FUNCTION_BLOCK "G302M_Code"
TITLE =G302M HEATING KILN 2
//COPYRIGHT:    (C) 2009  BUHLER AG, CH-9240 UZWIL, SWITZERLAND
//
//PRODUCT:      WinCoS_BIW01_09
//
//TITLE:        HEATING KILN 2
//                Machine group control
//                Maschinengruppensteuerung
//
//--------------------------------------------------------------------------------
//
//IDENT:        AUTHOR:             DEPT:                              DATE:
//
//P01_FB402.2.0 M.Wedler            AEB41                              27.Apr.2010
//             2nd Release
//P01_FB402.1.0 K.Renz              CSB41                              08.Okt.2009
//             1st Release
//
//--------------------------------------------------------------------------------
//
//PURPOSE:
//
//MANUAL :
//
//RESTRICTIONS:
//
//--------------------------------------------------------------------------------
AUTHOR : KR
FAMILY : USW
VERSION : 9.9


VAR
  Gr : "GCS7_GrpCtrlSub";	//Standard interface to group
  InOutValue1 : DINT ;	//Data for user
  InOutValue2 : DINT ;	//Data for user
  OutWayConflict : BOOL ;	//Data for user
  OutSelectionOk : BOOL ;	//Data for user
  CmdNewValue : BOOL ;	//Data for user
  CmdNewJob : BOOL ;	//Data for user
  OutCodeOK : BOOL ;	//Data for user
  InEndOfJob : BOOL ;	//Data for user
  staWayOk : BOOL ;	//Data for user
  EdgeStartRelease : BOOL ;	//Data for user
  USW8 : BOOL ;	//Data for user
  USW9 : BOOL ;	//Data for user
  USW10 : BOOL ;	//Data for user
  USW11 : BOOL ;	//Data for user
  USW12 : BOOL ;	//Data for user
  USW13 : BOOL ;	//Data for user
  USW14 : BOOL ;	//Data for user
  USW15 : BOOL ;	//Data for user
  A_3291_BPS21 : "GCS7_E_DigInput";	// DigInpCont
  A_3261_KCL11 : "GCS7_E_DigInput";	// DigInpCont
  A_3261_KCL11_AI : "GCS7_E_AnalogInput";	// AnaInp
  A_3261_KCL11_AO : "GCS7_E_AnalogOutput";	// AnaOutp
  A_3261_KCL11_EXT_ON : "GCS7_E_DigOutput";	// DigOut
  A_3261_KCL11_ON : "GCS7_E_DigInput";	// DigInpCont
  A_3261_KCL11_RUN : "GCS7_E_DigOutput";	// DigOut
  A_3261_KCL11_REG_ON : "GCS7_E_DigInput";	// DigInpCont
  A_3261_KCL11_REM_OP : "GCS7_E_DigInput";	// DigInpCont
END_VAR
VAR_TEMP
  tmpEnable : BOOL ;
  tmpFlag : BOOL ;
  tmpCmdNext : BOOL ;
  tmpLocal : BOOL ;
  tmpAspOk : BOOL ;
  tmpHWStop : BOOL ;
  tmpInstanzDBNo : INT ;
END_VAR
BEGIN
NETWORK
TITLE =



NETWORK
TITLE =Read command from group control
//Parameter
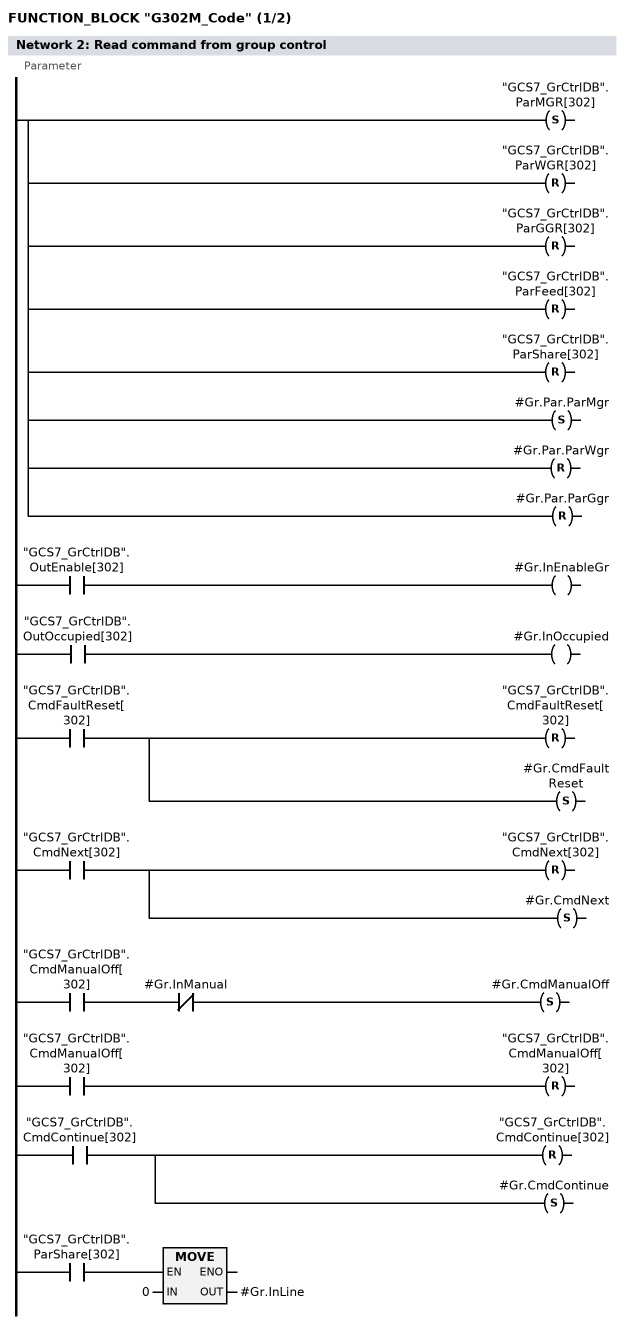
      SET   ;
      S     "GCS7_GrCtrlDB".ParMGR[302];
      R     "GCS7_GrCtrlDB".ParWGR[302];
      R     "GCS7_GrCtrlDB".ParGGR[302];
      R     "GCS7_GrCtrlDB".ParFeed[302];
      R     "GCS7_GrCtrlDB".ParShare[302];
      S     #Gr.Par.ParMgr;
      R     #Gr.Par.ParWgr;
      R     #Gr.Par.ParGgr;
//Command
      U     "GCS7_GrCtrlDB".OutEnable[302];
      =     #Gr.InEnableGr;
      U     "GCS7_GrCtrlDB".OutOccupied[302];
      =     #Gr.InOccupied;
      U     "GCS7_GrCtrlDB".CmdFaultReset[302];
      R     "GCS7_GrCtrlDB".CmdFaultReset[302];
      S     #Gr.CmdFaultReset;
      U     "GCS7_GrCtrlDB".CmdNext[302];
      R     "GCS7_GrCtrlDB".CmdNext[302];
      S     #Gr.CmdNext;

      U     "GCS7_GrCtrlDB".CmdManualOff[302];
      UN    #Gr.InManual;
      S     #Gr.CmdManualOff;
      U     "GCS7_GrCtrlDB".CmdManualOff[302];
      R     "GCS7_GrCtrlDB".CmdManualOff[302];

//      U     "GCS7_GrCtrlDB".CmdManualOff[302]
//      O     "GCS7_GrCtrlDB".OutOccupied[302]
//      R     "GCS7_GrCtrlDB".CmdManualOff[302]
//      S     #Gr.CmdManualOff

      U     "GCS7_GrCtrlDB".CmdContinue[302];
      R     "GCS7_GrCtrlDB".CmdContinue[302];
      S     #Gr.CmdContinue;
//Init Line Number
      U     "GCS7_GrCtrlDB".ParShare[302];
      SPBN  WE00;
      L     0;
      T     #Gr.InLine;
WE00: NOP   0;
NETWORK
TITLE =Call Methode Control
// 1. Handle Interface PCControl
// 2. Prepare mode --> ModePassive,ModeActive,ModeIdling
// 3. Reset global flags of the group
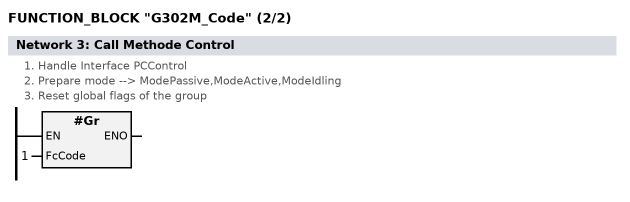
      CALL #Gr (
           FcCode                   := 1);
NETWORK
TITLE =Restart Idling Time

      L     #Gr.Par.ParIdling;
      L     2;
      >=I   ;
      SPB   IdTm;
      T     #Gr.Par.ParIdling;
IdTm: NOP   0;
      CLR   ;
      S     #Gr.CmdRestartIdling;
NETWORK
TITLE =Prepare global flags



NETWORK
TITLE =Set Pattern (Target position)

      U     #Gr.InManual;
      SPB   ILO6;
      L     "MAL1S033Par".StepAct.TemperaturBelowFloor;
      L     L#10;
      /D    ;
      DTR   ;
      U     "MAL1S033Par".Par.FlagProcess.Inf08; // Schritt halten
      SPBN  En06;
      L     "MAL1S033Par".RecipeHeader.SPARE_INT001; // Temp aus General Rezept
      DTR   ;
      SPA   En06;
ILO6: NOP   0;
      L     "MAL1S033Par".Par.ParIntProcess.TargetTemperature_ILO;
      ITD   ;
      DTR   ;
En06: T     "Regler Brenner 3".SP_INT; // setpoint temperature


NETWORK
TITLE =Interlocking WayOk

//BRT20100830 ====> Schritt abhängig den Abschaltpunkt für Brenner verändern
      U     "MAL1S033Par".Par.FlagProcess.ProcessActive;
      U(    ;
      L     "MAL1S033Par".Par.ParIntMachine.ActualStep;
      L     3;
      <I    ;
      )     ;
      U     "MAL1S032Par".Par.FlagProcess.Abdarr_Betrieb_Aktiv;
      L     "MAL1S033Par".StepAct.TemperaturBelowFloor;
      L     30;
      +I    ;
      L     10;
      *I    ;
      SPB   dif1;
      L     "MAL1S033Par".StepAct.TemperaturBelowFloor;
      L     100; // 10,0°C mehr als Sollwert
      +I    ;
      L     10;
      *I    ;
dif1: T     #InOutValue1; // Schaltpunkt für Brenner OFF

      U     "MAL1S033Par".Par.FlagProcess.ProcessActive;
      U(    ;
      L     "MAL1S033Par".Par.ParIntMachine.ActualStep;
      L     3;
      <I    ;
      )     ;
      U     "MAL1S032Par".Par.FlagProcess.Abdarr_Betrieb_Aktiv;
      L     "MAL1S033Par".StepAct.TemperaturBelowFloor;
      L     20;
      -I    ;
      L     10;
      *I    ;
      SPB   dif2;
      L     "MAL1S033Par".StepAct.TemperaturBelowFloor;
      L     10;
      *I    ;
dif2: T     #InOutValue2; // Schaltpunkt für Brenner ON


// Switch "OFF" Burner by Over Temperature
      U     "MAL1S033Par".Par.FlagProcess.ProcessActive;
      U(    ;
//      L     "MAL1S033Par".StepAct.TemperaturBelowFloor
//      L     100                         // 5,0°C mehr als Sollwert
//      +I
//      L     10
//      *I
      L     #InOutValue1; // Schaltpunkt für Brenner OFF
      L     "G295M".A_3291_BTE01.OutValuePc; //  Temperature Below Kiln Floor
      <=I   ;
      )     ;
      S     "G302M".USW8; //Over Temperature

      U(    ;
//      L     "MAL1S033Par".StepAct.TemperaturBelowFloor
//      L     10
//      *I
      L     #InOutValue2; // Schaltpunkt für Brenner ON
      L     "G295M".A_3291_BTE01.OutValuePc; //  Temperature Below Kiln Floor
      >=I   ;
      )     ;
      ON    "MAL1S033Par".Par.FlagProcess.ProcessActive;
      R     "G302M".USW8; //Over Temperature

//BRT20100830 <====
NETWORK
TITLE =Interlocking Autostart

      CLR   ;
      R     #Gr.OutAutostart;
NETWORK
TITLE =Interlocking Enable
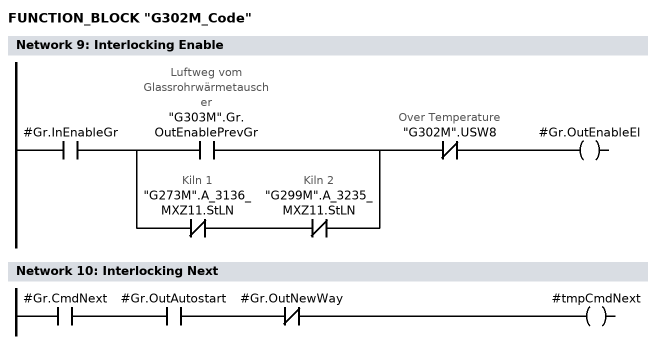

      U     #Gr.InEnableGr;
      U(    ;
      U     "G303M".Gr.OutEnablePrevGr; // Luftweg vom Glassrohrwärmetauscher
      O     ; // Umluftkanal
      UN    "G273M".A_3136_MXZ11.StLN; // Kiln 1
      UN    "G299M".A_3235_MXZ11.StLN; // Kiln 2
      )     ;
      UN    "G302M".USW8; //Over Temperature
      =     #Gr.OutEnableEl;

NETWORK
TITLE =Interlocking Next

      U     #Gr.CmdNext;
      U     #Gr.OutAutostart;
      UN    #Gr.OutNewWay;
      =     #tmpCmdNext;

NETWORK
TITLE =Interlocking Local / HWStop

      U     "PLC_SystemDB".GlobalFlags.Kilning_2;
      CLR   ;
      =     #tmpHWStop;

      U     #Gr.ModePassive;
      O     #tmpHWStop;
      =     #tmpLocal;

NETWORK
TITLE ==A-3291-BPS21 : HEAT EXCHANGE PRESSURE < 15mbar (Reserve)

      NOP   0;
//-InLocal---
      U     #tmpLocal;
      SET   ; // Nur einmal in Darre 1
      =     #A_3291_BPS21.InLocal;
//
//-Monitoring---
      CLR   ;
      =     #A_3291_BPS21.InMonTrue;
      CLR   ;
      =     #A_3291_BPS21.InMonFalse;
//
//-PreAlarm---
      CLR   ;
      =     #A_3291_BPS21.InPreAlarmTrue;
      CLR   ;
      =     #A_3291_BPS21.InPreAlarmFalse;
//
//-Additional commands---
//      CLR
//      S     #A_3291_BPS21.CmdRunTimeOutTime
//
//-Read inputs---
//      U     "A_3291_BPS21_I1"
      CLR   ;
      =     #A_3291_BPS21.InpTrue;
      U     "PLC_SystemDB".GlobalFlags.Kilning_2;
      =     #A_3291_BPS21.InHWStop;
      U     "PLC_DPInfo".Master[1].SlavesError[102];
      =     #A_3291_BPS21.InDPFault;
//
//-Set Parameters---
//
//-Call object control---
      CALL #A_3291_BPS21 ;
//
//-Write outputs---
NETWORK
TITLE ==A-3261-KCL11 : BURNER 3 ALARM SUMMARY

      NOP   0;
//-InLocal---
      U     #tmpLocal;
      =     #A_3261_KCL11.InLocal;
//
//-Monitoring---
      SET   ;
      =     #A_3261_KCL11.InMonTrue;
      CLR   ;
      =     #A_3261_KCL11.InMonFalse;
//
//-PreAlarm---
      CLR   ;
      =     #A_3261_KCL11.InPreAlarmTrue;
      CLR   ;
      =     #A_3261_KCL11.InPreAlarmFalse;
//
//-Additional commands---
//      CLR
//      S     #A_3261_KCL11.CmdRunTimeOutTime
//
//-Read inputs---
      UN    "A_3261_KCL11_I3";
      =     #A_3261_KCL11.InpTrue;
      U     "PLC_SystemDB".GlobalFlags.Kilning_2;
      =     #A_3261_KCL11.InHWStop;
      U     "PLC_DPInfo".Master[1].SlavesError[102];
      =     #A_3261_KCL11.InDPFault;
//
//-Set Parameters---
//
//-Call object control---
      CALL #A_3261_KCL11 ;
//
//-Write outputs---
NETWORK
TITLE ==A-3261-KCL11_EXT_ON : BURNER 3 EXTERAL ON
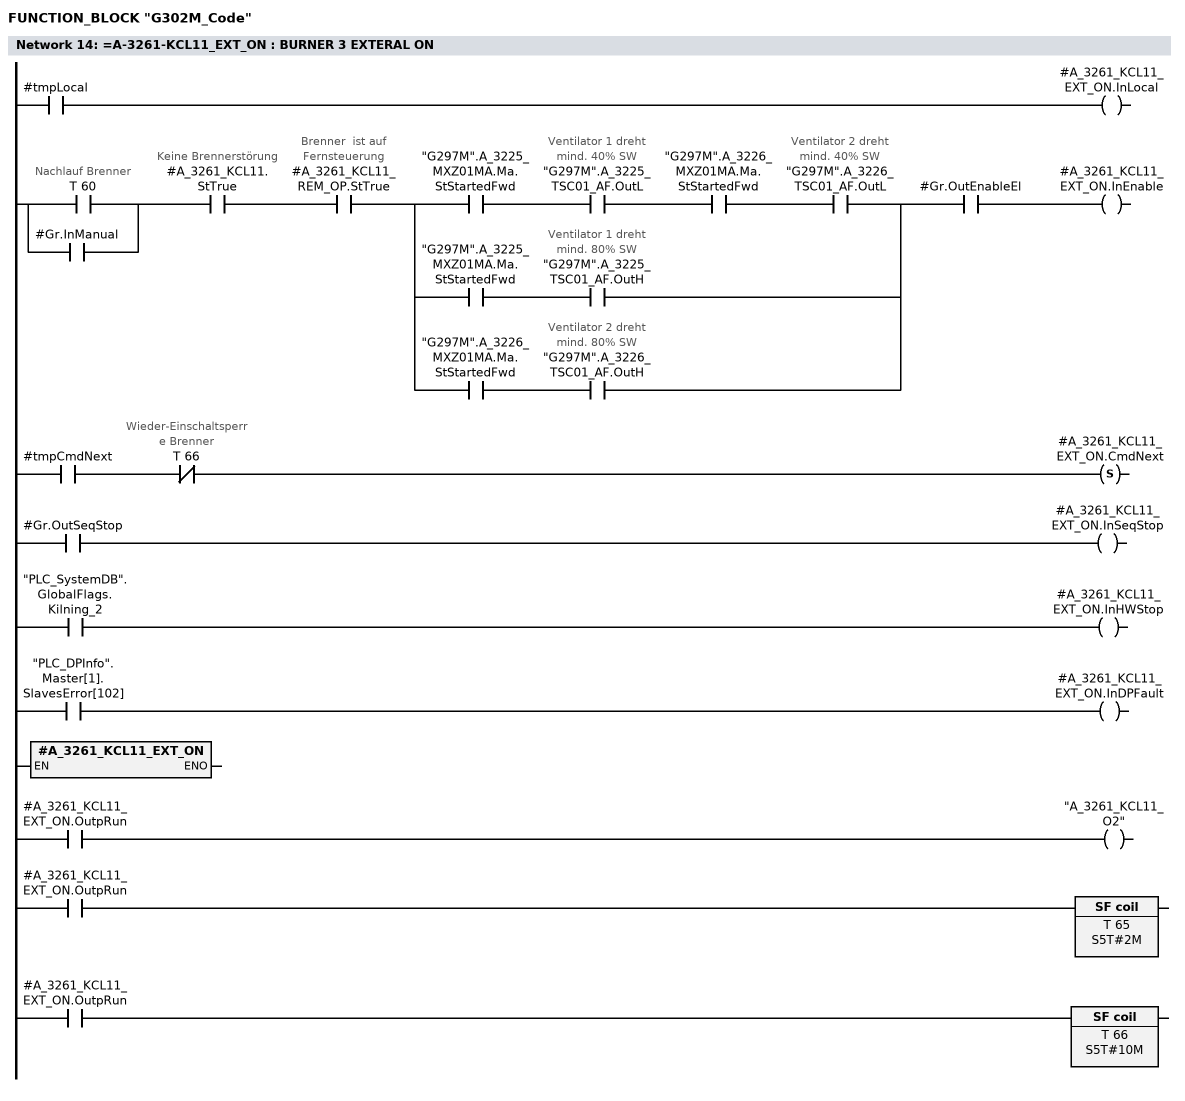

      NOP   0;
//-InLocal---
      U     #tmpLocal;
      =     #A_3261_KCL11_EXT_ON.InLocal;
//
//-Interlocking---
// Signal an Brenner 3: Start
      U     T     60; // Nachlauf Brenner
      O     #Gr.InManual;
      U     #A_3261_KCL11.StTrue; // Keine Brennerstörung
      U     #A_3261_KCL11_REM_OP.StTrue; // Brenner  ist auf Fernsteuerung
      U(    ;
      U     "G297M".A_3225_MXZ01MA.Ma.StStartedFwd;
      U     "G297M".A_3225_TSC01_AF.OutL; // Ventilator 1 dreht mind. 40% SW
      U     "G297M".A_3226_MXZ01MA.Ma.StStartedFwd;
      U     "G297M".A_3226_TSC01_AF.OutL; // Ventilator 2 dreht mind. 40% SW
      O     ;
      U(    ;
      U     "G297M".A_3225_MXZ01MA.Ma.StStartedFwd;
      U     "G297M".A_3225_TSC01_AF.OutH; // Ventilator 1 dreht mind. 80% SW
      O     ;
      U     "G297M".A_3226_MXZ01MA.Ma.StStartedFwd;
      U     "G297M".A_3226_TSC01_AF.OutH; // Ventilator 2 dreht mind. 80% SW
      )     ;
      )     ;
      U     #Gr.OutEnableEl;
      =     #A_3261_KCL11_EXT_ON.InEnable;
//
      U     #tmpCmdNext;
      UN    T     66; // Wieder-Einschaltsperre Brenner
      S     #A_3261_KCL11_EXT_ON.CmdNext;
//
      U     #Gr.OutSeqStop;
      =     #A_3261_KCL11_EXT_ON.InSeqStop;
//
//-Read inputs---
      U     "PLC_SystemDB".GlobalFlags.Kilning_2;
      =     #A_3261_KCL11_EXT_ON.InHWStop;
      U     "PLC_DPInfo".Master[1].SlavesError[102];
      =     #A_3261_KCL11_EXT_ON.InDPFault;
//
//-Set Parameters---
//
//-Call object control---
      CALL #A_3261_KCL11_EXT_ON ;
//
//-Write outputs---
      U     #A_3261_KCL11_EXT_ON.OutpRun;
      =     "A_3261_KCL11_O2";

      U     #A_3261_KCL11_EXT_ON.OutpRun;
      L     S5T#2M;
      SA    T     65; // Nachlauf Ventilator

// Um Stoerungen zu vermeiden
      U     #A_3261_KCL11_EXT_ON.OutpRun;
      L     S5T#10M;
      SA    T     66;

NETWORK
TITLE ==A-3261-KCL11_ON : BURNER 3 ON

      NOP   0;
//-InLocal---
      U     #tmpLocal;
      =     #A_3261_KCL11_ON.InLocal;
//
//-Monitoring---
      CLR   ;
      =     #A_3261_KCL11_ON.InMonTrue;
      CLR   ;
      =     #A_3261_KCL11_ON.InMonFalse;
//
//-PreAlarm---
      CLR   ;
      =     #A_3261_KCL11_ON.InPreAlarmTrue;
      CLR   ;
      =     #A_3261_KCL11_ON.InPreAlarmFalse;
//
//-Additional commands---
//      CLR
//      S     #A_3261_KCL11_ON.CmdRunTimeOutTime
//
//-Read inputs---
      U     "A_3261_KCL11_I1";
      =     #A_3261_KCL11_ON.InpTrue;
      U     "PLC_SystemDB".GlobalFlags.Kilning_2;
      =     #A_3261_KCL11_ON.InHWStop;
      U     "PLC_DPInfo".Master[1].SlavesError[102];
      =     #A_3261_KCL11_ON.InDPFault;
//
//-Set Parameters---
//
//-Call object control---
      CALL #A_3261_KCL11_ON ;
//
//-Write outputs---
NETWORK
TITLE ==A-3261-KCL11_RUN : BURNER 3 MAIN FAN RUNNING
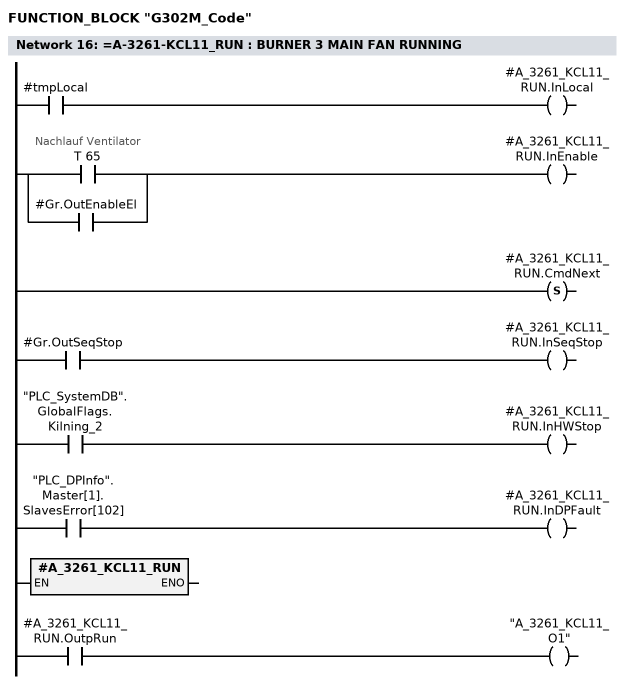

      NOP   0;
//-InLocal---
      U     #tmpLocal;
      =     #A_3261_KCL11_RUN.InLocal;
//
//-Interlocking---
      U     T     65; // Nachlauf Ventilator
      O     #Gr.OutEnableEl;
      =     #A_3261_KCL11_RUN.InEnable;
//
      SET   ;
      S     #A_3261_KCL11_RUN.CmdNext;
//
      U     #Gr.OutSeqStop;
      =     #A_3261_KCL11_RUN.InSeqStop;
//
//-Read inputs---
      U     "PLC_SystemDB".GlobalFlags.Kilning_2;
      =     #A_3261_KCL11_RUN.InHWStop;
      U     "PLC_DPInfo".Master[1].SlavesError[102];
      =     #A_3261_KCL11_RUN.InDPFault;
//
//-Set Parameters---
//
//-Call object control---
      CALL #A_3261_KCL11_RUN ;
//
//-Write outputs---
      U     #A_3261_KCL11_RUN.OutpRun;
      =     "A_3261_KCL11_O1";

NETWORK
TITLE ==A-3261-KCL11_AI : BURNER 3 INPUT SIGNAL ANALOG

      NOP   0;
//-InLocal---
      U     #tmpLocal;
      SET   ;
      =     #A_3261_KCL11_AI.InLocal;

//-Monitoring---
      CLR   ;
      =     #A_3261_KCL11_AI.InMonLL;
      CLR   ;
      =     #A_3261_KCL11_AI.InMonL;
      CLR   ;
      =     #A_3261_KCL11_AI.InMonMid;
      CLR   ;
      =     #A_3261_KCL11_AI.InMonH;
      CLR   ;
      =     #A_3261_KCL11_AI.InMonHH;
//
//-Read inputs---
      L     "A_3261_KCL11_AI1";
// Negative Werte ignorieren
      L     0;
      <I    ;
      SPB   v017;
      TAK   ;
v017: T     #A_3261_KCL11_AI.InpValue;

      U     "PLC_SystemDB".GlobalFlags.Kilning_2;
      =     #A_3261_KCL11_AI.InHWStop;
      U     "PLC_DPInfo".Master[1].SlavesError[102];
      =     #A_3261_KCL11_AI.InDPFault;
//
//-Set Parameters---
//
//-Call object control---
      CALL #A_3261_KCL11_AI ;
//
//-Write outputs---
NETWORK
TITLE ==A-3261-KCL11_AO : BURNER 3 OUTPUT SIGNAL ANALOG

      NOP   0;
//-InLocal---
      U     #tmpLocal;
      =     #A_3261_KCL11_AO.InLocal;

//-Interlocking---
      CLR   ;
      =     #A_3261_KCL11_AO.InDisable;

//-Values and parameters---
      L     "Regler Brenner 3".LMN_PER;
      T     #A_3261_KCL11_AO.InOutValuePc;
      T     "A_3261_KCL11_AO1";
//
//-Read inputs---
      U     "PLC_SystemDB".GlobalFlags.Kilning_2;
      =     #A_3261_KCL11_AO.InHWStop;
      U     "PLC_DPInfo".Master[1].SlavesError[102];
      =     #A_3261_KCL11_AO.InDPFault;
//
//-Set Parameters---
//
//-Call object control---
      CALL #A_3261_KCL11_AO ;
//
//-Write outputs---
//      L     #A_3261_KCL11_AO.OutpValue
//      T     "A_3261_KCL11_AO1"
//      UN    "PLC_SystemDB".TestFunctions.StaIOSimuli
//      SPB   PA0
//      T     AW  1028
//PA0:  NOP   0
NETWORK
TITLE ==A-3261-KCL11_REG_ON : BURNER 3 REGULATOR ON

      NOP   0;
//-InLocal---
      U     #tmpLocal;
      =     #A_3261_KCL11_REG_ON.InLocal;
//
//-Monitoring---
      CLR   ;
      =     #A_3261_KCL11_REG_ON.InMonTrue;
      CLR   ;
      =     #A_3261_KCL11_REG_ON.InMonFalse;
//
//-PreAlarm---
      CLR   ;
      =     #A_3261_KCL11_REG_ON.InPreAlarmTrue;
      CLR   ;
      =     #A_3261_KCL11_REG_ON.InPreAlarmFalse;
//
//-Additional commands---
//      CLR
//      S     #A_3261_KCL11_REG_ON.CmdRunTimeOutTime
//
//-Read inputs---
      U     "A_3261_KCL11_I2";
      =     #A_3261_KCL11_REG_ON.InpTrue;
      U     "PLC_SystemDB".GlobalFlags.Kilning_2;
      =     #A_3261_KCL11_REG_ON.InHWStop;
      U     "PLC_DPInfo".Master[1].SlavesError[102];
      =     #A_3261_KCL11_REG_ON.InDPFault;
//
//-Set Parameters---
//
//-Call object control---
      CALL #A_3261_KCL11_REG_ON ;
//
//-Write outputs---
NETWORK
TITLE ==A-3261-KCL11_REM_OP : BURNER 3 REMOTE OPERATION

      NOP   0;
//-InLocal---
      U     #tmpLocal;
      =     #A_3261_KCL11_REM_OP.InLocal;
//
//-Monitoring---
      SET   ;
      =     #A_3261_KCL11_REM_OP.InMonTrue;
      CLR   ;
      =     #A_3261_KCL11_REM_OP.InMonFalse;
//
//-PreAlarm---
      CLR   ;
      =     #A_3261_KCL11_REM_OP.InPreAlarmTrue;
      CLR   ;
      =     #A_3261_KCL11_REM_OP.InPreAlarmFalse;
//
//-Additional commands---
//      CLR
//      S     #A_3261_KCL11_REM_OP.CmdRunTimeOutTime
//
//-Read inputs---
      U     "A_3261_KCL11_I4";
      =     #A_3261_KCL11_REM_OP.InpTrue;
      U     "PLC_SystemDB".GlobalFlags.Kilning_2;
      =     #A_3261_KCL11_REM_OP.InHWStop;
      U     "PLC_DPInfo".Master[1].SlavesError[102];
      =     #A_3261_KCL11_REM_OP.InDPFault;
//
//-Set Parameters---
//
//-Call object control---
      CALL #A_3261_KCL11_REM_OP ;
//
//-Write outputs---
NETWORK
TITLE =Test Fault
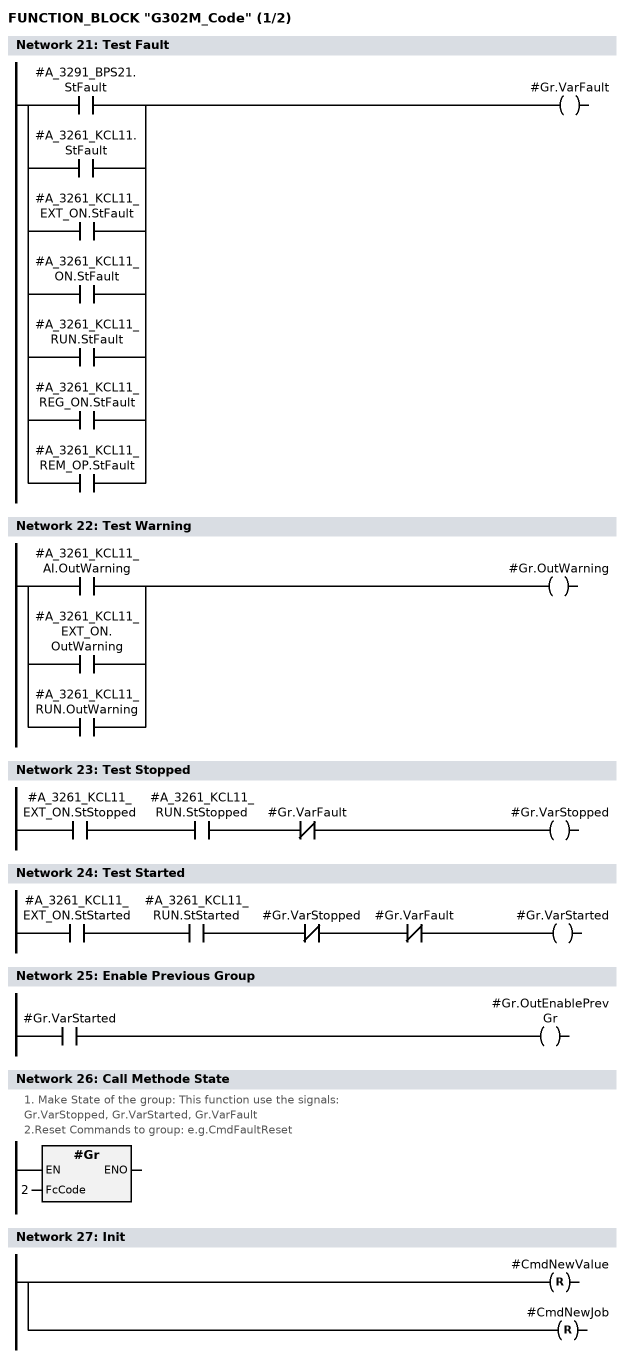

      U     #A_3291_BPS21.StFault;
      O     #A_3261_KCL11.StFault;
//      O     #A_3261_KCL11_AI.OutFaulted
//      O     #A_3261_KCL11_AO.StFault
      O     #A_3261_KCL11_EXT_ON.StFault;
      O     #A_3261_KCL11_ON.StFault;
      O     #A_3261_KCL11_RUN.StFault;
      O     #A_3261_KCL11_REG_ON.StFault;
      O     #A_3261_KCL11_REM_OP.StFault;
      =     #Gr.VarFault;
NETWORK
TITLE =Test Warning

      U     #A_3261_KCL11_AI.OutWarning;
      O     #A_3261_KCL11_EXT_ON.OutWarning;
      O     #A_3261_KCL11_RUN.OutWarning;
      =     #Gr.OutWarning;
NETWORK
TITLE =Test Stopped

      U     #A_3261_KCL11_EXT_ON.StStopped;
      U     #A_3261_KCL11_RUN.StStopped;
      UN    #Gr.VarFault;
      =     #Gr.VarStopped;
NETWORK
TITLE =Test Started

      U     #A_3261_KCL11_EXT_ON.StStarted;
      U     #A_3261_KCL11_RUN.StStarted;
      UN    #Gr.VarStopped;
      UN    #Gr.VarFault;
      =     #Gr.VarStarted;
NETWORK
TITLE =Enable Previous Group

      U     #Gr.VarStarted;
      =     #Gr.OutEnablePrevGr;
NETWORK
TITLE =Call Methode State
//1. Make State of the group: This function use the signals:
//        Gr.VarStopped, Gr.VarStarted, Gr.VarFault
//2.Reset Commands to group: e.g.CmdFaultReset
      CALL #Gr (
           FcCode                   := 2);
NETWORK
TITLE =Init

      SET   ;
      R     #CmdNewValue;
      R     #CmdNewJob;
NETWORK
TITLE =Write data to group control
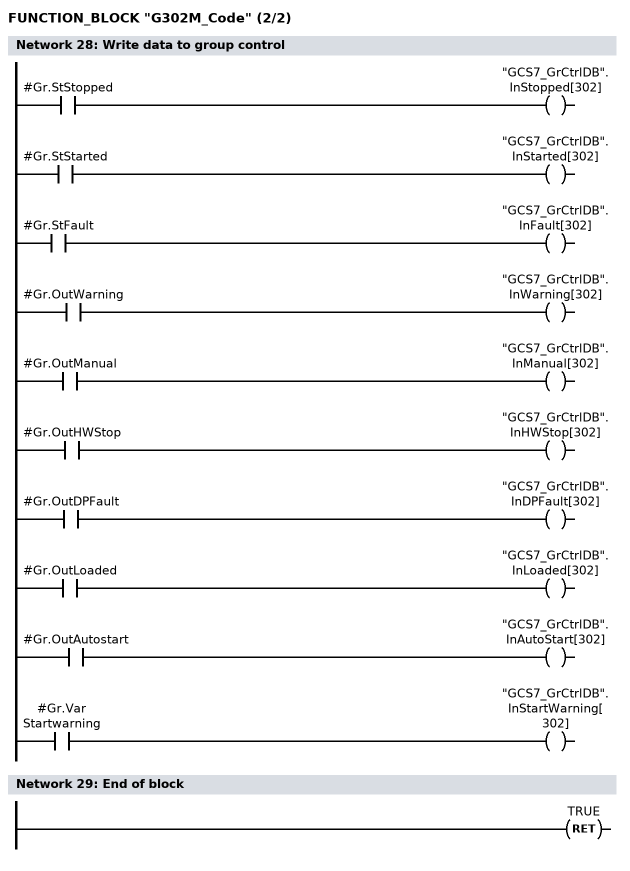

      U     #Gr.StStopped;
      =     "GCS7_GrCtrlDB".InStopped[302];
      U     #Gr.StStarted;
      =     "GCS7_GrCtrlDB".InStarted[302];
      U     #Gr.StFault;
      =     "GCS7_GrCtrlDB".InFault[302];
      U     #Gr.OutWarning;
      =     "GCS7_GrCtrlDB".InWarning[302];
      U     #Gr.OutManual;
      =     "GCS7_GrCtrlDB".InManual[302];
      U     #Gr.OutHWStop;
      =     "GCS7_GrCtrlDB".InHWStop[302];
      U     #Gr.OutDPFault;
      =     "GCS7_GrCtrlDB".InDPFault[302];
      U     #Gr.OutLoaded;
      =     "GCS7_GrCtrlDB".InLoaded[302];
      U     #Gr.OutAutostart;
      =     "GCS7_GrCtrlDB".InAutoStart[302];
      U     #Gr.VarStartwarning;
      =     "GCS7_GrCtrlDB".InStartWarning[302];
NETWORK
TITLE =End of block

      BE    ;

END_FUNCTION_BLOCK

